(* PLC project Recipe_Tool, Beckhoff Automation GmbH TwinCAT PLC Control 3.5.3.40 *)
(* stored: creationDateTime 2014-11-23T04:17:58.5837056, modificationDateTime 2014-11-23T04:17:58.5837056 *)

FUNCTION_BLOCK Recipe_10053_911Targa
  VAR_INPUT
    execute : BOOL;
    Order : DUT_RECIPEORDER;
  END_VAR
  VAR_OUTPUT
    RecipeInfo : DUT_RECIPEOFFER;
    RecipeDone : BOOL;
    InitDone : BOOL;
    Ready : BOOL;
  END_VAR
  VAR
    userparametersum : LREAL;
    StepDone : BOOL;
    i : INT;
    Command : ARRAY[1..5] OF DUT_RecipeCommand;
    NextSkill : BOOL;
    SectionReady : BOOL;
  END_VAR

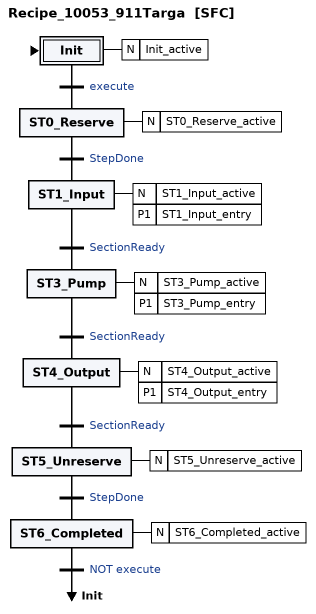
INITIAL_STEP Init:
  Init_active(N);
END_STEP
TRANSITION FROM Init TO ST0_Reserve
  := execute;
END_TRANSITION
STEP ST0_Reserve:
  ST0_Reserve_active(N);
END_STEP
TRANSITION FROM ST0_Reserve TO ST1_Input
  := StepDone;
END_TRANSITION
STEP ST1_Input:
  ST1_Input_active(N);
  ST1_Input_entry(P1);
END_STEP
TRANSITION FROM ST1_Input TO ST3_Pump
  := SectionReady;
END_TRANSITION
STEP ST3_Pump:
  ST3_Pump_active(N);
  ST3_Pump_entry(P1);
END_STEP
TRANSITION FROM ST3_Pump TO ST4_Output
  := SectionReady;
END_TRANSITION
STEP ST4_Output:
  ST4_Output_active(N);
  ST4_Output_entry(P1);
END_STEP
TRANSITION FROM ST4_Output TO ST5_Unreserve
  := SectionReady;
END_TRANSITION
STEP ST5_Unreserve:
  ST5_Unreserve_active(N);
END_STEP
TRANSITION FROM ST5_Unreserve TO ST6_Completed
  := StepDone;
END_TRANSITION
STEP ST6_Completed:
  ST6_Completed_active(N);
END_STEP
TRANSITION FROM ST6_Completed TO Init
  := NOT execute;
END_TRANSITION

ACTION Init_active:
                //RT: 2014.11.23: Vorbereiten der daten und der HMI
RecipeDone := FALSE;

// Initialisation of Recipe Parameters an name etc
RecipeInfo.Name := '911 Targa';
RecipeInfo.Description := '';
RecipeInfo.Dummy := FALSE;
RecipeInfo.RecipeID := 10053; 	// 
Initdone := TRUE;

Command[1].SkillID := 1113;
Command[1].SkillName := 'Maracuja Juice';
Command[1].Quantity := 29;

Command[2].SkillID := 1117;
Command[2].SkillName := 'Orange Juice';
Command[2].Quantity := 29;

Command[3].SkillID := 1114;
Command[3].SkillName := 'Pineapple Juice';
Command[3].Quantity := 29;

Command[4].SkillID := 1112;
Command[4].SkillName := 'Citrone Juice';
Command[4].Quantity := 14;

Command[5].SkillID := 1111;
Command[5].SkillName := 'Grenadine Syrup';
Command[5].Quantity := 14;

//Parameter 0:

	RecipeInfo.UserParameter[0].Dummy 		:= FALSE;
	RecipeInfo.UserParameter[0].Default		:= 200;
	RecipeInfo.UserParameter[0].Description	:= 'Gives the total fluid amount in the glass';
	RecipeInfo.UserParameter[0].MaxValue	:= 200;
	RecipeInfo.UserParameter[0].MinValue	:= 10;
	RecipeInfo.UserParameter[0].Name		:= 'Total Liquid Amount';
	RecipeInfo.UserParameter[0].Unit		:= 'ml';
	
//Parameter 1-5:
FOR i := 1 TO 5 DO
	IF Command[i].SkillID = 0 THEN
		RecipeInfo.UserParameter[i].Dummy 		:= TRUE;
	ELSE
		RecipeInfo.UserParameter[i].Dummy 		:= FALSE;
		RecipeInfo.UserParameter[i].Default		:= Command[i].Quantity;
		RecipeInfo.UserParameter[i].Description	:= Command[i].SkillName;
		RecipeInfo.UserParameter[i].MaxValue	:= 100;
		RecipeInfo.UserParameter[i].MinValue	:= 1;
		RecipeInfo.UserParameter[i].Name		:= Command[i].SkillName;
		RecipeInfo.UserParameter[i].Unit		:= 'ml';	
	END_IF
END_FOR

              
END_ACTION

ACTION ST1_Input_active:
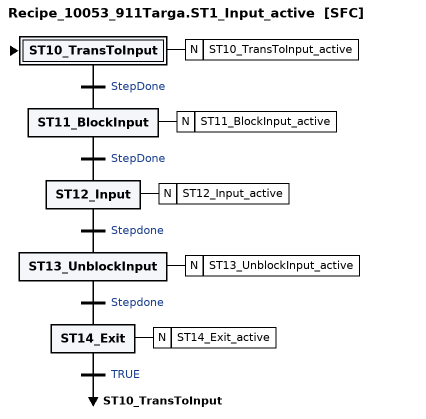
INITIAL_STEP ST10_TransToInput:
  ST10_TransToInput_active(N);
END_STEP
TRANSITION FROM ST10_TransToInput TO ST11_BlockInput
  := StepDone;
END_TRANSITION
STEP ST11_BlockInput:
  ST11_BlockInput_active(N);
END_STEP
TRANSITION FROM ST11_BlockInput TO ST12_Input
  := StepDone;
END_TRANSITION
STEP ST12_Input:
  ST12_Input_active(N);
END_STEP
TRANSITION FROM ST12_Input TO ST13_UnblockInput
  := Stepdone;
END_TRANSITION
STEP ST13_UnblockInput:
  ST13_UnblockInput_active(N);
END_STEP
TRANSITION FROM ST13_UnblockInput TO ST14_Exit
  := Stepdone;
END_TRANSITION
STEP ST14_Exit:
  ST14_Exit_active(N);
END_STEP
TRANSITION FROM ST14_Exit TO ST10_TransToInput
  := TRUE;
END_TRANSITION
END_ACTION

ACTION ST1_Reserve0_active:
                //RT: 2014.11.23: Reservire einen Mover

StepDone := FALSE;
RecipeDone := FALSE;
//Skill auswählen
ExecuteSkill.SkillID 		:= 1310;
ExecuteSkill.SkillName	 	:= 'Reserve';

//Parameter setzen

ExecuteSkill.Parameter[1].ID := 1;
ExecuteSkill.Parameter[1].Name := 'TaskID';
ExecuteSkill.Parameter[1].Value := Order.TaskID;

(*
ExecuteSkill.Parameter[2].ID := ;
ExecuteSkill.Parameter[2].Name := '';
ExecuteSkill.Parameter[2].Value := ;
*)

(*
ExecuteSkill.Parameter[3].ID := ;
ExecuteSkill.Parameter[3].Name := '';
ExecuteSkill.Parameter[3].Value := ;
*)

(*
ExecuteSkill.Parameter[4].ID := ;
ExecuteSkill.Parameter[4].Name := '';
ExecuteSkill.Parameter[4].Value := ;
*)

(*
ExecuteSkill.Parameter[5].ID := ;
ExecuteSkill.Parameter[5].Name := '';
ExecuteSkill.Parameter[5].Value := ;
*)

ExecuteSkill();

StepDone := ExecuteSkill.Done;
              
END_ACTION

ACTION ST10_TransToInput_active:
                //RT: 2014.11.23: Mover zum Input

StepDone := FALSE;

//Skill auswählen
ExecuteSkill.SkillID 		:= 1320;
ExecuteSkill.SkillName	 	:= 'Transport';

//Parameter setzen

ExecuteSkill.Parameter[3].ID := 3;
ExecuteSkill.Parameter[3].Name := 'Velocity';
ExecuteSkill.Parameter[3].Value := 1000;



ExecuteSkill.Parameter[1].ID :=  1;
ExecuteSkill.Parameter[1].Name := 'TargetPosition X';
ExecuteSkill.Parameter[1].Value := 30 ;
ExecuteSkill.Parameter[1].StringValue := '#DP#2#XPosition';



ExecuteSkill.Parameter[2].ID := 2;
ExecuteSkill.Parameter[2].Name := 'TargetPosition Z';
ExecuteSkill.Parameter[2].Value := 100;// ZCookieModule - ZCookieModuleCalibration - 2* Cookiethickness + toppingthickness+ Preasureheight  ;



(*
ExecuteSkill.Parameter[4].ID := 4;
ExecuteSkill.Parameter[4].Name := 'Acceleration';
ExecuteSkill.Parameter[4].Value := 0 ;
*)

(*
ExecuteSkill.Parameter[5].ID := ;
ExecuteSkill.Parameter[5].Name := '';
ExecuteSkill.Parameter[5].Value := ;
*)



ExecuteSkill();

StepDone := ExecuteSkill.Done;
              
END_ACTION

ACTION ST11_BlockInput_active:
                //RT: 2014.11.23: Blockirt den Mover an Position
StepDone := FALSE;

//Skill auswählen
ExecuteSkill.SkillID 		:= 1315;
ExecuteSkill.SkillName	 	:= 'Block';

//Parameter setzen

ExecuteSkill.Parameter[1].ID := 1;
ExecuteSkill.Parameter[1].Name := 'TaskID';
ExecuteSkill.Parameter[1].Value := Order.TaskID;


(*
ExecuteSkill.Parameter[2].ID := ;
ExecuteSkill.Parameter[2].Name := '';
ExecuteSkill.Parameter[2].Value := ;
*)

(*
ExecuteSkill.Parameter[3].ID := ;
ExecuteSkill.Parameter[3].Name := '';
ExecuteSkill.Parameter[3].Value := ;
*)

(*
ExecuteSkill.Parameter[4].ID := ;
ExecuteSkill.Parameter[4].Name := '';
ExecuteSkill.Parameter[4].Value := ;
*)

(*
ExecuteSkill.Parameter[5].ID := ;
ExecuteSkill.Parameter[5].Name := '';
ExecuteSkill.Parameter[5].Value := ;
*)



ExecuteSkill();

StepDone := ExecuteSkill.Done;
              
END_ACTION

ACTION ST1_Input_entry:
                SectionReady := FALSE;

              
END_ACTION

ACTION ST0_Reserve_active:
                //RT: 2014.11.23: Reservire einen Mover

StepDone := FALSE;
RecipeDone := FALSE;
//Skill auswählen
ExecuteSkill.SkillID 		:= 1310;
ExecuteSkill.SkillName	 	:= 'Reserve';

//Parameter setzen

ExecuteSkill.Parameter[1].ID := 1;
ExecuteSkill.Parameter[1].Name := 'TaskID';
ExecuteSkill.Parameter[1].Value := Order.TaskID;

(*
ExecuteSkill.Parameter[2].ID := ;
ExecuteSkill.Parameter[2].Name := '';
ExecuteSkill.Parameter[2].Value := ;
*)

(*
ExecuteSkill.Parameter[3].ID := ;
ExecuteSkill.Parameter[3].Name := '';
ExecuteSkill.Parameter[3].Value := ;
*)

(*
ExecuteSkill.Parameter[4].ID := ;
ExecuteSkill.Parameter[4].Name := '';
ExecuteSkill.Parameter[4].Value := ;
*)

(*
ExecuteSkill.Parameter[5].ID := ;
ExecuteSkill.Parameter[5].Name := '';
ExecuteSkill.Parameter[5].Value := ;
*)

ExecuteSkill();

StepDone := ExecuteSkill.Done;
              
END_ACTION

ACTION ST12_Input_active:
                //RT: 2014.11.23: Input Modul auslösen
StepDone := FALSE;

//Skill auswählen
ExecuteSkill.SkillID 		:= 1402;
ExecuteSkill.SkillName	 	:= 'Input';

//Parameter setzen

ExecuteSkill.Parameter[1].ID := 1;
ExecuteSkill.Parameter[1].Name := 'TaskID';
ExecuteSkill.Parameter[1].Value := Order.TaskID;


(*
ExecuteSkill.Parameter[2].ID := ;
ExecuteSkill.Parameter[2].Name := '';
ExecuteSkill.Parameter[2].Value := ;
*)

(*
ExecuteSkill.Parameter[3].ID := ;
ExecuteSkill.Parameter[3].Name := '';
ExecuteSkill.Parameter[3].Value := ;
*)

(*
ExecuteSkill.Parameter[4].ID := ;
ExecuteSkill.Parameter[4].Name := '';
ExecuteSkill.Parameter[4].Value := ;
*)

(*
ExecuteSkill.Parameter[5].ID := ;
ExecuteSkill.Parameter[5].Name := '';
ExecuteSkill.Parameter[5].Value := ;
*)



ExecuteSkill();

StepDone := ExecuteSkill.Done;
              
END_ACTION

ACTION ST13_UnblockInput_active:
                //RT: 2014.11.23: Gibt Mover Position Frei
StepDone := FALSE;

//Skill auswählen
ExecuteSkill.SkillID 		:= 1316;
ExecuteSkill.SkillName	 	:= 'Unblock';

//Parameter setzen

ExecuteSkill.Parameter[1].ID := 1;
ExecuteSkill.Parameter[1].Name := 'TaskID';
ExecuteSkill.Parameter[1].Value := Order.TaskID;


(*
ExecuteSkill.Parameter[2].ID := ;
ExecuteSkill.Parameter[2].Name := '';
ExecuteSkill.Parameter[2].Value := ;
*)

(*
ExecuteSkill.Parameter[3].ID := ;
ExecuteSkill.Parameter[3].Name := '';
ExecuteSkill.Parameter[3].Value := ;
*)

(*
ExecuteSkill.Parameter[4].ID := ;
ExecuteSkill.Parameter[4].Name := '';
ExecuteSkill.Parameter[4].Value := ;
*)

(*
ExecuteSkill.Parameter[5].ID := ;
ExecuteSkill.Parameter[5].Name := '';
ExecuteSkill.Parameter[5].Value := ;
*)



ExecuteSkill();

StepDone := ExecuteSkill.Done;
              
END_ACTION

ACTION ST14_Exit_active:
                SectionReady := TRUE;
              
END_ACTION

ACTION ST3_Pump_active:
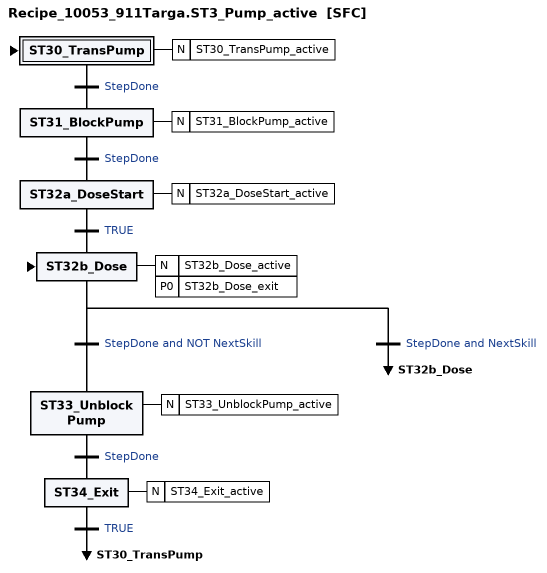
INITIAL_STEP ST30_TransPump:
  ST30_TransPump_active(N);
END_STEP
TRANSITION FROM ST30_TransPump TO ST31_BlockPump
  := StepDone;
END_TRANSITION
STEP ST31_BlockPump:
  ST31_BlockPump_active(N);
END_STEP
TRANSITION FROM ST31_BlockPump TO ST32a_DoseStart
  := StepDone;
END_TRANSITION
STEP ST32a_DoseStart:
  ST32a_DoseStart_active(N);
END_STEP
TRANSITION FROM ST32a_DoseStart TO ST32b_Dose
  := TRUE;
END_TRANSITION
STEP ST32b_Dose:
  ST32b_Dose_active(N);
  ST32b_Dose_exit(P0);
END_STEP
TRANSITION FROM ST32b_Dose TO ST33_UnblockPump
  := StepDone and NOT NextSkill;
END_TRANSITION
TRANSITION FROM ST32b_Dose TO ST32b_Dose
  := StepDone and NextSkill;
END_TRANSITION
STEP ST33_UnblockPump:
  ST33_UnblockPump_active(N);
END_STEP
TRANSITION FROM ST33_UnblockPump TO ST34_Exit
  := StepDone;
END_TRANSITION
STEP ST34_Exit:
  ST34_Exit_active(N);
END_STEP
TRANSITION FROM ST34_Exit TO ST30_TransPump
  := TRUE;
END_TRANSITION
END_ACTION

ACTION ST3_Pump_entry:
                SectionReady := FALSE;
              
END_ACTION

ACTION ST30_TransPump_active:
                //RT: 2014.11.23: Mover zum Pump
StepDone := FALSE;

//Skill auswählen
ExecuteSkill.SkillID 		:= 1320;
ExecuteSkill.SkillName	 	:= 'Transport';

//Parameter setzen

ExecuteSkill.Parameter[3].ID := 3;
ExecuteSkill.Parameter[3].Name := 'Velocity';
ExecuteSkill.Parameter[3].Value := 1000;



ExecuteSkill.Parameter[1].ID :=  1;
ExecuteSkill.Parameter[1].Name := 'TargetPosition X';
ExecuteSkill.Parameter[1].Value := 30 ;
ExecuteSkill.Parameter[1].StringValue := '#DP#2#XPosition';



ExecuteSkill.Parameter[2].ID := 2;
ExecuteSkill.Parameter[2].Name := 'TargetPosition Z';
ExecuteSkill.Parameter[2].Value := 10;// ZCookieModule - ZCookieModuleCalibration - 2* Cookiethickness + toppingthickness+ Preasureheight  ;



(*
ExecuteSkill.Parameter[4].ID := 4;
ExecuteSkill.Parameter[4].Name := 'Acceleration';
ExecuteSkill.Parameter[4].Value := 0 ;
*)

(*
ExecuteSkill.Parameter[5].ID := ;
ExecuteSkill.Parameter[5].Name := '';
ExecuteSkill.Parameter[5].Value := ;
*)



ExecuteSkill();

StepDone := ExecuteSkill.Done;
              
END_ACTION

ACTION ST31_BlockPump_active:
                //RT: 2014.11.23: Blockirt den Mover an Position
StepDone := FALSE;

//Skill auswählen
ExecuteSkill.SkillID 		:= 1315;
ExecuteSkill.SkillName	 	:= 'Block';

//Parameter setzen

ExecuteSkill.Parameter[1].ID := 1;
ExecuteSkill.Parameter[1].Name := 'TaskID';
ExecuteSkill.Parameter[1].Value := Order.TaskID;


(*
ExecuteSkill.Parameter[2].ID := ;
ExecuteSkill.Parameter[2].Name := '';
ExecuteSkill.Parameter[2].Value := ;
*)

(*
ExecuteSkill.Parameter[3].ID := ;
ExecuteSkill.Parameter[3].Name := '';
ExecuteSkill.Parameter[3].Value := ;
*)

(*
ExecuteSkill.Parameter[4].ID := ;
ExecuteSkill.Parameter[4].Name := '';
ExecuteSkill.Parameter[4].Value := ;
*)

(*
ExecuteSkill.Parameter[5].ID := ;
ExecuteSkill.Parameter[5].Name := '';
ExecuteSkill.Parameter[5].Value := ;
*)



ExecuteSkill();

StepDone := ExecuteSkill.Done;
              
END_ACTION

ACTION ST34_Exit_active:
                SectionReady := TRUE;
              
END_ACTION

ACTION ST33_UnblockPump_active:
                //RT: 2014.11.23: Gibt Mover Position Frei
StepDone := FALSE;

//Skill auswählen
ExecuteSkill.SkillID 		:= 1316;
ExecuteSkill.SkillName	 	:= 'Unblock';

//Parameter setzen

ExecuteSkill.Parameter[1].ID := 1;
ExecuteSkill.Parameter[1].Name := 'TaskID';
ExecuteSkill.Parameter[1].Value := Order.TaskID;


(*
ExecuteSkill.Parameter[2].ID := ;
ExecuteSkill.Parameter[2].Name := '';
ExecuteSkill.Parameter[2].Value := ;
*)

(*
ExecuteSkill.Parameter[3].ID := ;
ExecuteSkill.Parameter[3].Name := '';
ExecuteSkill.Parameter[3].Value := ;
*)

(*
ExecuteSkill.Parameter[4].ID := ;
ExecuteSkill.Parameter[4].Name := '';
ExecuteSkill.Parameter[4].Value := ;
*)

(*
ExecuteSkill.Parameter[5].ID := ;
ExecuteSkill.Parameter[5].Name := '';
ExecuteSkill.Parameter[5].Value := ;
*)



ExecuteSkill();

StepDone := ExecuteSkill.Done;
              
END_ACTION

ACTION ST32b_Dose_active:
                //RT: 2014.11.23: Die Dosir Skills anlegen
StepDone := FALSE;

//Skill auswählen
ExecuteSkill.SkillID 		:= Command[i].SkillID;
ExecuteSkill.SkillName	 	:= Command[i].SkillName;
//Parameter setzen

ExecuteSkill.Parameter[0].ID := 1;
ExecuteSkill.Parameter[0].Name := 'Quantity';
//order.userParameter[0] = amount
ExecuteSkill.Parameter[0].Value := order.UserParameter[0].Value * order.UserParameter[i].Value / userparametersum ;//Summe aller Zutatenmengen;

(*
ExecuteSkill.Parameter[2].ID := ;
ExecuteSkill.Parameter[2].Name := '';
ExecuteSkill.Parameter[2].Value := ;
*)

(*
ExecuteSkill.Parameter[3].ID := ;
ExecuteSkill.Parameter[3].Name := '';
ExecuteSkill.Parameter[3].Value := ;
*)

(*
ExecuteSkill.Parameter[4].ID := ;
ExecuteSkill.Parameter[4].Name := '';
ExecuteSkill.Parameter[4].Value := ;
*)

(*
ExecuteSkill.Parameter[5].ID := ;
ExecuteSkill.Parameter[5].Name := '';
ExecuteSkill.Parameter[5].Value := ;
*)


ExecuteSkill();

StepDone := ExecuteSkill.Done;

              
END_ACTION

ACTION ST32b_Dose_exit:
                i := i + 1 ;

IF i = 6 THEN
	NextSkill := FALSE;
ELSIF Command[i + 1].SkillID = 0 THEN
	NextSkill := FALSE;
ELSE
	NextSkill := TRUE;
END_IF


              
END_ACTION

ACTION ST32a_DoseStart_active:
                //RT: 2014.11.23: Summe aller zutaten zum Normiren

userparametersum := 0;
FOR i := 1 TO UserParameterCnt DO
	IF NOT (order.UserParameter[i].Value = 0) THEN
		userparametersum := userparametersum + order.UserParameter[i].Value;
	
	END_IF
END_FOR
IF userparametersum = 0 THEN
userparametersum := -1;
END_IF

//RT: 2014.11.23: Start wert des Arrays setzen
i := 1;
              
END_ACTION

ACTION ST4_Output_active:
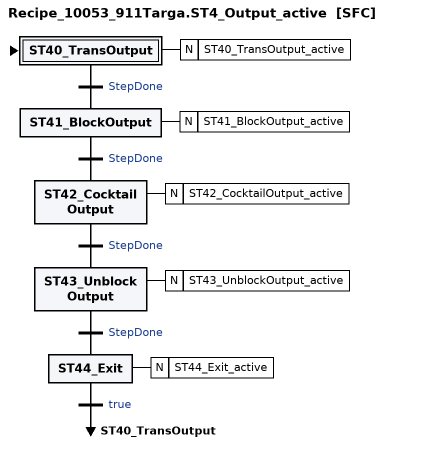
INITIAL_STEP ST40_TransOutput:
  ST40_TransOutput_active(N);
END_STEP
TRANSITION FROM ST40_TransOutput TO ST41_BlockOutput
  := StepDone;
END_TRANSITION
STEP ST41_BlockOutput:
  ST41_BlockOutput_active(N);
END_STEP
TRANSITION FROM ST41_BlockOutput TO ST42_CocktailOutput
  := StepDone;
END_TRANSITION
STEP ST42_CocktailOutput:
  ST42_CocktailOutput_active(N);
END_STEP
TRANSITION FROM ST42_CocktailOutput TO ST43_UnblockOutput
  := StepDone;
END_TRANSITION
STEP ST43_UnblockOutput:
  ST43_UnblockOutput_active(N);
END_STEP
TRANSITION FROM ST43_UnblockOutput TO ST44_Exit
  := StepDone;
END_TRANSITION
STEP ST44_Exit:
  ST44_Exit_active(N);
END_STEP
TRANSITION FROM ST44_Exit TO ST40_TransOutput
  := true;
END_TRANSITION
END_ACTION

ACTION ST4_Output_entry:
                SectionReady := FALSE;
              
END_ACTION

ACTION ST40_TransOutput_active:
                //RT: 2014.11.23: Mover zum Output
StepDone := FALSE;

//Skill auswählen
ExecuteSkill.SkillID 		:= 1320;
ExecuteSkill.SkillName	 	:= 'Transport';

//Parameter setzen

ExecuteSkill.Parameter[3].ID := 3;
ExecuteSkill.Parameter[3].Name := 'Velocity';
ExecuteSkill.Parameter[3].Value := 300;



ExecuteSkill.Parameter[1].ID :=  1;
ExecuteSkill.Parameter[1].Name := 'TargetPosition X';
ExecuteSkill.Parameter[1].Value := 30 ;
ExecuteSkill.Parameter[1].StringValue := '#DP#2#XPosition';



ExecuteSkill.Parameter[2].ID := 2;
ExecuteSkill.Parameter[2].Name := 'TargetPosition Z';
ExecuteSkill.Parameter[2].Value := 100;// ZCookieModule - ZCookieModuleCalibration - 2* Cookiethickness + toppingthickness+ Preasureheight  ;



(* ExecuteSkill.Parameter[4].ID := 4;
ExecuteSkill.Parameter[4].Name := 'Acceleration';
ExecuteSkill.Parameter[4].Value :=0 ;

*)
(*
ExecuteSkill.Parameter[5].ID := ;
ExecuteSkill.Parameter[5].Name := '';
ExecuteSkill.Parameter[5].Value := ;
*)



ExecuteSkill();

StepDone := ExecuteSkill.Done;
              
END_ACTION

ACTION ST41_BlockOutput_active:
                //RT: 2014.11.23: Blockirt den Mover an Position
StepDone := FALSE;

//Skill auswählen
ExecuteSkill.SkillID 		:= 1315;
ExecuteSkill.SkillName	 	:= 'Block';

//Parameter setzen

ExecuteSkill.Parameter[1].ID := 1;
ExecuteSkill.Parameter[1].Name := 'TaskID';
ExecuteSkill.Parameter[1].Value := Order.TaskID;


(*
ExecuteSkill.Parameter[2].ID := ;
ExecuteSkill.Parameter[2].Name := '';
ExecuteSkill.Parameter[2].Value := ;
*)

(*
ExecuteSkill.Parameter[3].ID := ;
ExecuteSkill.Parameter[3].Name := '';
ExecuteSkill.Parameter[3].Value := ;
*)

(*
ExecuteSkill.Parameter[4].ID := ;
ExecuteSkill.Parameter[4].Name := '';
ExecuteSkill.Parameter[4].Value := ;
*)

(*
ExecuteSkill.Parameter[5].ID := ;
ExecuteSkill.Parameter[5].Name := '';
ExecuteSkill.Parameter[5].Value := ;
*)



ExecuteSkill();

StepDone := ExecuteSkill.Done;
              
END_ACTION

ACTION ST42_CocktailOutput_active:
                //RT: 2014.11.23: Ausgeben des Produktes
StepDone := FALSE;

//Skill auswählen
ExecuteSkill.SkillID 		:= 1403;
ExecuteSkill.SkillName	 	:= 'Output';

//Parameter setzen

ExecuteSkill.Parameter[1].ID := 1;
ExecuteSkill.Parameter[1].Name := 'TaskID';
ExecuteSkill.Parameter[1].Value := Order.TaskID;


(*
ExecuteSkill.Parameter[2].ID := ;
ExecuteSkill.Parameter[2].Name := '';
ExecuteSkill.Parameter[2].Value := ;
*)

(*
ExecuteSkill.Parameter[3].ID := ;
ExecuteSkill.Parameter[3].Name := '';
ExecuteSkill.Parameter[3].Value := ;
*)

(*
ExecuteSkill.Parameter[4].ID := ;
ExecuteSkill.Parameter[4].Name := '';
ExecuteSkill.Parameter[4].Value := ;
*)

(*
ExecuteSkill.Parameter[5].ID := ;
ExecuteSkill.Parameter[5].Name := '';
ExecuteSkill.Parameter[5].Value := ;
*)



ExecuteSkill();

StepDone := ExecuteSkill.Done;
              
END_ACTION

ACTION ST43_UnblockOutput_active:
                //RT: 2014.11.23: Gibt Mover Position Frei
StepDone := FALSE;

//Skill auswählen
ExecuteSkill.SkillID 		:= 1316;
ExecuteSkill.SkillName	 	:= 'Unblock';

//Parameter setzen

ExecuteSkill.Parameter[1].ID := 1;
ExecuteSkill.Parameter[1].Name := 'TaskID';
ExecuteSkill.Parameter[1].Value := Order.TaskID;


(*
ExecuteSkill.Parameter[2].ID := ;
ExecuteSkill.Parameter[2].Name := '';
ExecuteSkill.Parameter[2].Value := ;
*)

(*
ExecuteSkill.Parameter[3].ID := ;
ExecuteSkill.Parameter[3].Name := '';
ExecuteSkill.Parameter[3].Value := ;
*)

(*
ExecuteSkill.Parameter[4].ID := ;
ExecuteSkill.Parameter[4].Name := '';
ExecuteSkill.Parameter[4].Value := ;
*)

(*
ExecuteSkill.Parameter[5].ID := ;
ExecuteSkill.Parameter[5].Name := '';
ExecuteSkill.Parameter[5].Value := ;
*)



ExecuteSkill();

StepDone := ExecuteSkill.Done;
              
END_ACTION

ACTION ST44_Exit_active:
                SectionReady := TRUE;
              
END_ACTION

ACTION ST5_Unreserve_active:
                //RT: 2014.11.23: Mover Freigeben
StepDone := FALSE;

//Skill auswählen
ExecuteSkill.SkillID 		:= 1311;
ExecuteSkill.SkillName	 	:= 'Unreserve';

//Parameter setzen

ExecuteSkill.Parameter[1].ID := 1;
ExecuteSkill.Parameter[1].Name := 'TaskID';
ExecuteSkill.Parameter[1].Value := Order.TaskID;


(*
ExecuteSkill.Parameter[2].ID := ;
ExecuteSkill.Parameter[2].Name := '';
ExecuteSkill.Parameter[2].Val ue := ;
*)

(*
ExecuteSkill.Parameter[3].ID := ;
ExecuteSkill.Parameter[3].Name := '';
ExecuteSkill.Parameter[3].Value := ;
*)

(*
ExecuteSkill.Parameter[4].ID := ;
ExecuteSkill.Parameter[4].Name := '';
ExecuteSkill.Parameter[4].Value := ;
*)

(*
ExecuteSkill.Parameter[5].ID := ;
ExecuteSkill.Parameter[5].Name := '';
ExecuteSkill.Parameter[5].Value := ;
*)



ExecuteSkill();

StepDone := ExecuteSkill.Done;
              
END_ACTION

ACTION ST6_Completed_active:
                //RT: 2014.11.23: Warte auf Execute = False
RecipeDone := TRUE;
StepDone := FALSE;
              
END_ACTION
END_FUNCTION_BLOCK
